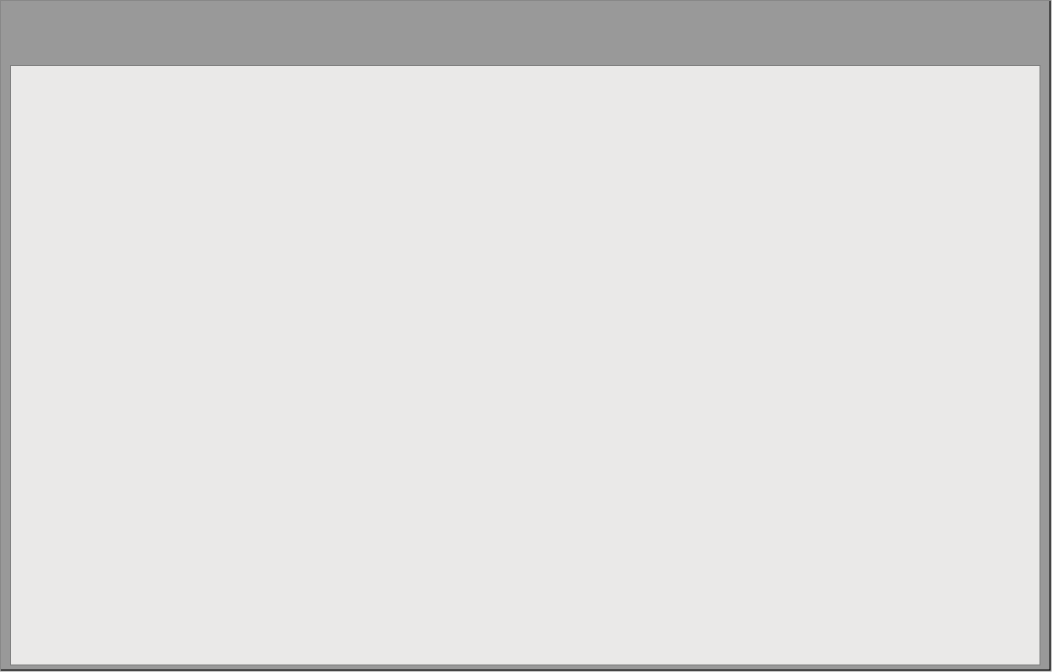
VISUALIZATION VISU_SystemBackground  // 1052x672
VAR_IN_OUT
	color : StatusColor;
END_VAR
    Rectangle (0,0 1050x670)
        p3450524324: color.bg
    Rectangle (10,65 1030x600)
END_VISUALIZATION

(* stored: Version 1.1.0.1, ProductVersion 3.1.4018.2
   Visu VISU_SystemBackground: Id {d924cdab-e870-4893-a6ca-fe37801c0458} *)
